FUNCTION_BLOCK DataPanel_MI_IX (* Input service interface function block for boolean input data *)
  (* Description: Copyright (c) 2014, 2015 fortiss GmbH, HR Agrartechnik GmbH This program and the accompanying materials are made available under the terms of the Eclipse Public License 2.0 which is available at https://www.eclipse.org/legal/epl-2.0/ SPDX-License-Identifier: EPL-2.0 *)
  (* Version 1.0, 2014-08-26, Waldemar Eisenmenger, fortiss GmbH, initial API and implementation and/or initial documentation *)
  (* Version 1.1, 2014-08-30, Alois Zoitl, fortiss GmbH *)
  (* Version 1.2, 2015-06-10, Monika Wenger, fortiss GmbH *)
  PACKAGE DataPanel::io::MI::DI;
  IMPORT DataPanel::io::MI::const::MI;
  IMPORT eclipse4diac::core::TypeHash;
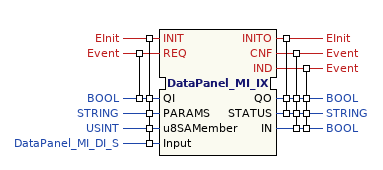
  EVENT_INPUT
    INIT : EInit WITH QI, PARAMS, u8SAMember, Input; (* Service Initialization *)
    REQ WITH QI; (* Service Request *)
  END_EVENT
  EVENT_OUTPUT
    INITO : EInit WITH QO, STATUS; (* Initialization Confirm *)
    CNF WITH QO, STATUS, IN; (* Confirmation of Requested Service *)
    IND WITH QO, STATUS, IN; (* Indication from Resource *)
  END_EVENT
  VAR_INPUT
    QI : BOOL; (* Event Input Qualifier *)
    PARAMS : STRING; (* Service Parameters *)
    u8SAMember : USINT := MI::MI_00; (* Node SA 224..239 *)
    Input : DataPanel::io::MI::DI::DataPanel_MI_DI_S := DataPanel_MI_DI::Invalid; (* Identify the Input DigitalInput_5A..8B *)
  END_VAR
  VAR_OUTPUT
    QO : BOOL; (* Event Output Qualifier *)
    STATUS : STRING; (* Service Status *)
    IN : BOOL; (* Input data from resource *)
  END_VAR
END_FUNCTION_BLOCK
